# EPICS autosave request: iocBoot/ioc13bmd_LVP_XPS/auto_settings.req
file "CARS_motor_settings.req",         P=$(P), M=m97
file "CARS_motor_settings.req",         P=$(P), M=m98
file "CARS_motor_settings.req",         P=$(P), M=m99
file "CARS_motor_settings.req",         P=$(P), M=m100
file "CARS_motor_settings.req",         P=$(P), M=m101
file "CARS_motor_settings.req",         P=$(P), M=m102
file "CARS_motor_settings.req",         P=$(P), M=m103
file "CARS_motor_settings.req",         P=$(P), M=m104
